KUKA KRL data list: test.dat

&ACCESS RVP
&REL 3
&PARAM DISKPATH = KRC:\R1\Program\JUZI\AAA
DEFDAT  test
   ;FOLD EXTERNAL DECLARATIONS;%{PE}%MKUKATPBASIS,%CEXT,%VCOMMON,%P
   ;FOLD BASISTECH EXT;%{PE}%MKUKATPBASIS,%CEXT,%VEXT,%P
   EXT  BAS (BAS_COMMAND  :IN,REAL  :IN )
   DECL INT SUCCESS
   ;ENDFOLD (BASISTECH EXT)
   ;FOLD USER EXT;%{E}%MKUKATPUSER,%CEXT,%VEXT,%P
   ;Make your modifications here

   ;ENDFOLD (USER EXT)
   ;ENDFOLD (EXTERNAL DECLARATIONS)

   INT RST, nLen
   DECL CHAR strMsg[256], LOG_MSG[2047]

ENDDAT
